INTERFACE I_LightTower

END_INTERFACE

(* stored: Version 1.1.0.1, ProductVersion 3.1.4024.13
   Itf I_LightTower: Id {fc793eea-f426-0d8b-312b-328114c2bcfb} *)
